# EPICS autosave request: soft_iocs/galil_DMC/iocBoot/iocgalil_DMC_E02/slit_settings.req
file "2slit_soft_settings.req", P=$(P), SLIT=JJ_C_V:
file "2slit_soft_settings.req", P=$(P), SLIT=JJ_C_H:
